(* CoDeSys 2.3 export: PARAMETERMENU_TS.EXP *)

(* Data type in Diag/Parameter *)
TYPE ParameterMenu_ts :
STRUCT
	MenuName_as8			: STRING(32);
(*	MenuName_as8			: ARRAY [1..4] OF STRING(32);*)
	ParameterGroup_as		: ARRAY [1..8] OF ParameterGroup_ts;
END_STRUCT
END_TYPE
